TYPE "UDT_MEStoPLC_ext"
VERSION : 0.1
   STRUCT
      Cmd : Struct
         "MES.Load_PartOK" : Bool;
         "MES.Load_PartNG" : Bool;
         "MES.Load_2" : Bool;
         "MES.Load_3" : Bool;
         "MES.Unload_DataSaveOK" : Bool;
         "MES.Unload_DataSaveNOK" : Bool;
         "MES.Unload_2" : Bool;
         "MES.Unload_3" : Bool;
         "MES.Spare8" : Bool;
         "MES.Spare9" : Bool;
         "MES.Spare10" : Bool;
         "MES.Spare11" : Bool;
         "MES.Spare12" : Bool;
         "MES.Spare13" : Bool;
         "MES.Spare14" : Bool;
         "MES.HeartbeatSignal" : Bool;
      END_STRUCT;
   END_STRUCT;

END_TYPE

